PROGRAM MAIN
VAR
	test : DINT;
END_VAR

test := test + 4;

END_PROGRAM

(* stored: Version 1.1.0.1
   POU MAIN: Id {d218bcac-1e7f-436c-b85f-5bd99c1d019c}, SpecialFunc None *)
